ORGANIZATION_BLOCK "Main"
{ S7_Optimized_Access := 'TRUE' }
VERSION : 1.0
BEGIN
   "FC_BagPulseDustCollector_IO"();
END_ORGANIZATION_BLOCK
